// TIA Portal V17 export
// export: Created 2024-08-26T21:07:15.2242134Z, ExportSetting WithDefaults, DisplayName Totally Integrated Automation Portal, DisplayVersion V17 Update 7, DisplayName TIA Portal Openness, DisplayVersion V17 Update 7, DisplayName TIA Portal Version Control Interface, DisplayVersion V17, DisplayName SINAMICS Startdrive Advanced, DisplayVersion V17 SP2, DisplayName SINAMICS Startdrive G110M, G120, G120C, G120D, G120P, G115D, DisplayVersion V17 SP2, DisplayName SINAMICS Startdrive G130, G150, S120, S150, SINAMICS MV, S210, DisplayVersion V17 SP2, DisplayName STEP 7 Professional, DisplayVersion V17 Update 7, DisplayName STEP 7 Safety, DisplayVersion V17 Update 6, DisplayName WinCC Advanced / Unified PC, DisplayVersion V17 Update 7
ORGANIZATION_BLOCK "stationOutputs"   // OB124, LAD, ProgramCycle
TITLE = "Main Program Sweep (Cycle)"
{ S7_Optimized_Access := 'TRUE' }
VERSION : 0.1
// stored: AutoNumber true, IsIECCheckEnabled false, SetENOAutomatically false
   VAR_INPUT
      Initial_Call : Bool;   // Initial call of this OB
      Remanence : Bool;   // =True, if remanent data are available
   END_VAR
BEGIN

REGION Network 1: PRESENT PARTS
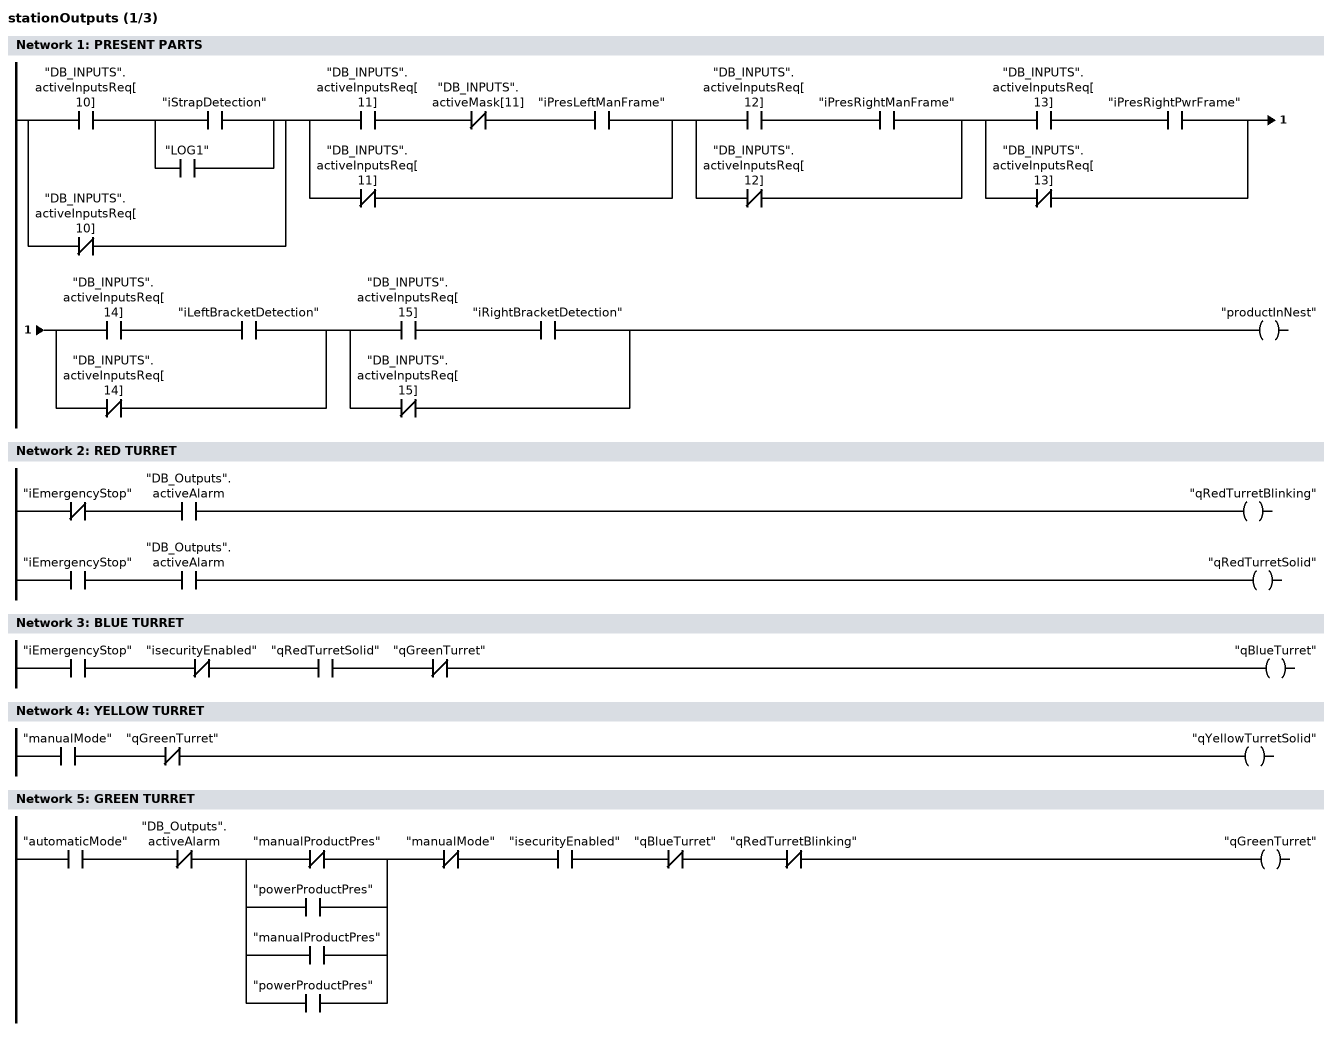
   RUNG wire#powerrail
      Contact( "DB_INPUTS".activeInputsReq[10] )
      wire#w1
      Contact( "iStrapDetection" )
      wire#w2
      Contact( "DB_INPUTS".activeInputsReq[11] )
      I_Contact( "DB_INPUTS".activeMask[11] )
      Contact( "iPresLeftManFrame" )
      wire#w3
      Contact( "DB_INPUTS".activeInputsReq[12] )
      Contact( "iPresRightManFrame" )
      wire#w4
      Contact( "DB_INPUTS".activeInputsReq[13] )
      Contact( "iPresRightPwrFrame" )
      wire#w5
      Contact( "DB_INPUTS".activeInputsReq[14] )
      Contact( "iLeftBracketDetection" )
      wire#w6
      Contact( "DB_INPUTS".activeInputsReq[15] )
      Contact( "iRightBracketDetection" )
      wire#w7
      Coil( "productInNest" )
   END_RUNG
   RUNG wire#w1
      Contact( "LOG1" )
   END_RUNG wire#w2
   RUNG wire#powerrail
      I_Contact( "DB_INPUTS".activeInputsReq[10] )
   END_RUNG wire#w2
   RUNG wire#w2
      I_Contact( "DB_INPUTS".activeInputsReq[11] )
   END_RUNG wire#w3
   RUNG wire#w3
      I_Contact( "DB_INPUTS".activeInputsReq[12] )
   END_RUNG wire#w4
   RUNG wire#w4
      I_Contact( "DB_INPUTS".activeInputsReq[13] )
   END_RUNG wire#w5
   RUNG wire#w5
      I_Contact( "DB_INPUTS".activeInputsReq[14] )
   END_RUNG wire#w6
   RUNG wire#w6
      I_Contact( "DB_INPUTS".activeInputsReq[15] )
   END_RUNG wire#w7
   // the same network as SCL:
   "productInNest" := (("DB_INPUTS".activeInputsReq[10] AND ("iStrapDetection" OR "LOG1")) OR NOT "DB_INPUTS".activeInputsReq[10]) AND (("DB_INPUTS".activeInputsReq[11] AND NOT "DB_INPUTS".activeMask[11] AND "iPresLeftManFrame") OR NOT "DB_INPUTS".activeInputsReq[11]) AND (("DB_INPUTS".activeInputsReq[12] AND "iPresRightManFrame") OR NOT "DB_INPUTS".activeInputsReq[12]) AND (("DB_INPUTS".activeInputsReq[13] AND "iPresRightPwrFrame") OR NOT "DB_INPUTS".activeInputsReq[13]) AND (("DB_INPUTS".activeInputsReq[14] AND "iLeftBracketDetection") OR NOT "DB_INPUTS".activeInputsReq[14]) AND (("DB_INPUTS".activeInputsReq[15] AND "iRightBracketDetection") OR NOT "DB_INPUTS".activeInputsReq[15]);
END_REGION

REGION Network 2: RED TURRET
   RUNG wire#powerrail
      I_Contact( "iEmergencyStop" )
      Contact( "DB_Outputs".activeAlarm )
      Coil( "qRedTurretBlinking" )
   END_RUNG
   RUNG wire#powerrail
      Contact( "iEmergencyStop" )
      Contact( "DB_Outputs".activeAlarm )
      Coil( "qRedTurretSolid" )
   END_RUNG
   // the same network as SCL:
   "qRedTurretBlinking" := NOT "iEmergencyStop" AND "DB_Outputs".activeAlarm;
   "qRedTurretSolid" := "iEmergencyStop" AND "DB_Outputs".activeAlarm;
END_REGION

REGION Network 3: BLUE TURRET
   RUNG wire#powerrail
      Contact( "iEmergencyStop" )
      I_Contact( "isecurityEnabled" )
      Contact( "qRedTurretSolid" )
      I_Contact( "qGreenTurret" )
      Coil( "qBlueTurret" )
   END_RUNG
   // the same network as SCL:
   "qBlueTurret" := "iEmergencyStop" AND NOT "isecurityEnabled" AND "qRedTurretSolid" AND NOT "qGreenTurret";
END_REGION

REGION Network 4: YELLOW TURRET
   RUNG wire#powerrail
      Contact( "manualMode" )
      I_Contact( "qGreenTurret" )
      Coil( "qYellowTurretSolid" )
   END_RUNG
   // the same network as SCL:
   "qYellowTurretSolid" := "manualMode" AND NOT "qGreenTurret";
END_REGION

REGION Network 5: GREEN TURRET
   RUNG wire#powerrail
      Contact( "automaticMode" )
      I_Contact( "DB_Outputs".activeAlarm )
      wire#w1
      I_Contact( "manualProductPres" )
      wire#w2
      I_Contact( "manualMode" )
      Contact( "isecurityEnabled" )
      I_Contact( "qBlueTurret" )
      I_Contact( "qRedTurretBlinking" )
      Coil( "qGreenTurret" )
   END_RUNG
   RUNG wire#w1
      Contact( "powerProductPres" )
   END_RUNG wire#w2
   RUNG wire#w1
      Contact( "manualProductPres" )
   END_RUNG wire#w2
   RUNG wire#w1
      Contact( "powerProductPres" )
   END_RUNG wire#w2
   // the same network as SCL:
   "qGreenTurret" := "automaticMode" AND NOT "DB_Outputs".activeAlarm AND (NOT "manualProductPres" OR "powerProductPres" OR "manualProductPres" OR "powerProductPres") AND NOT "manualMode" AND "isecurityEnabled" AND NOT "qBlueTurret" AND NOT "qRedTurretBlinking";
END_REGION

REGION Network 6: SmartLight
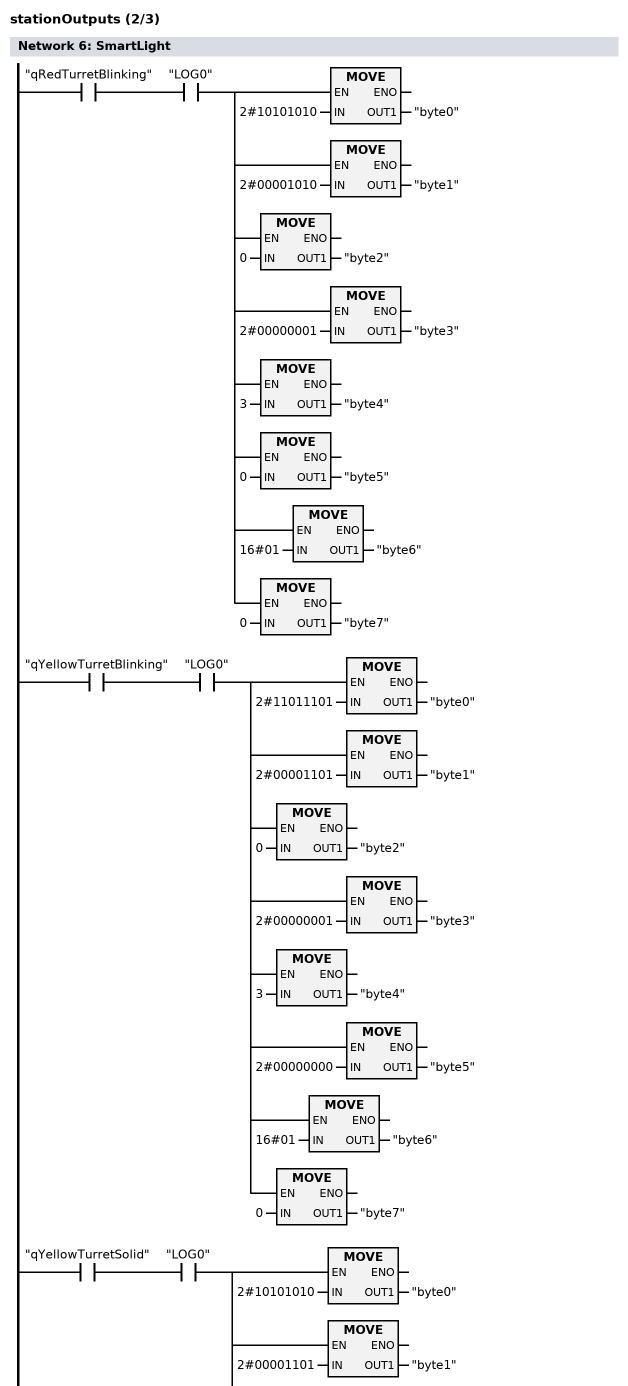
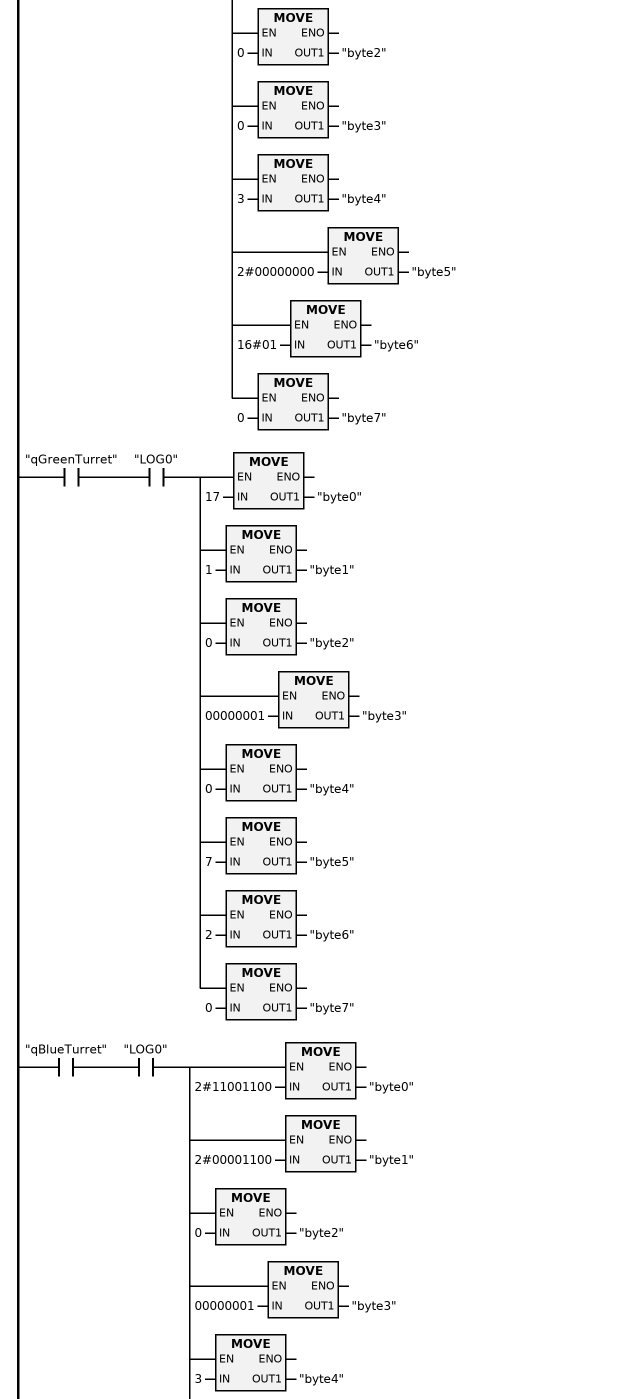
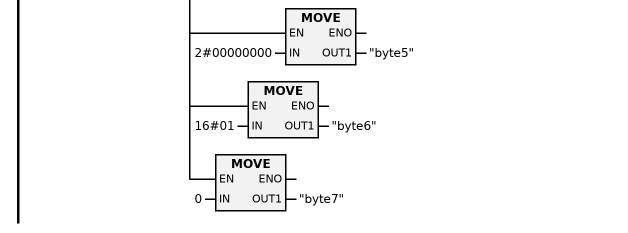
   RUNG wire#powerrail
      Contact( "qRedTurretBlinking" )
      Contact( "LOG0" )
      wire#w1
      Move(in := 2#10101010, out1 => "byte0")
   END_RUNG
   RUNG wire#w1
      Move(in := 2#00001010, out1 => "byte1")
   END_RUNG
   RUNG wire#w1
      Move(in := 0, out1 => "byte2")
   END_RUNG
   RUNG wire#w1
      Move(in := 2#00000001, out1 => "byte3")
   END_RUNG
   RUNG wire#w1
      Move(in := 3, out1 => "byte4")
   END_RUNG
   RUNG wire#w1
      Move(in := 0, out1 => "byte5")
   END_RUNG
   RUNG wire#w1
      Move(in := 16#01, out1 => "byte6")
   END_RUNG
   RUNG wire#w1
      Move(in := 0, out1 => "byte7")
   END_RUNG
   RUNG wire#powerrail
      Contact( "qYellowTurretBlinking" )
      Contact( "LOG0" )
      wire#w2
      Move(in := 2#11011101, out1 => "byte0")
   END_RUNG
   RUNG wire#w2
      Move(in := 2#00001101, out1 => "byte1")
   END_RUNG
   RUNG wire#w2
      Move(in := 0, out1 => "byte2")
   END_RUNG
   RUNG wire#w2
      Move(in := 2#00000001, out1 => "byte3")
   END_RUNG
   RUNG wire#w2
      Move(in := 3, out1 => "byte4")
   END_RUNG
   RUNG wire#w2
      Move(in := 2#00000000, out1 => "byte5")
   END_RUNG
   RUNG wire#w2
      Move(in := 16#01, out1 => "byte6")
   END_RUNG
   RUNG wire#w2
      Move(in := 0, out1 => "byte7")
   END_RUNG
   RUNG wire#powerrail
      Contact( "qYellowTurretSolid" )
      Contact( "LOG0" )
      wire#w3
      Move(in := 2#10101010, out1 => "byte0")
   END_RUNG
   RUNG wire#w3
      Move(in := 2#00001101, out1 => "byte1")
   END_RUNG
   RUNG wire#w3
      Move(in := 0, out1 => "byte2")
   END_RUNG
   RUNG wire#w3
      Move(in := 0, out1 => "byte3")
   END_RUNG
   RUNG wire#w3
      Move(in := 3, out1 => "byte4")
   END_RUNG
   RUNG wire#w3
      Move(in := 2#00000000, out1 => "byte5")
   END_RUNG
   RUNG wire#w3
      Move(in := 16#01, out1 => "byte6")
   END_RUNG
   RUNG wire#w3
      Move(in := 0, out1 => "byte7")
   END_RUNG
   RUNG wire#powerrail
      Contact( "qGreenTurret" )
      Contact( "LOG0" )
      wire#w4
      Move(in := 17, out1 => "byte0")
   END_RUNG
   RUNG wire#w4
      Move(in := 1, out1 => "byte1")
   END_RUNG
   RUNG wire#w4
      Move(in := 0, out1 => "byte2")
   END_RUNG
   RUNG wire#w4
      Move(in := 00000001, out1 => "byte3")
   END_RUNG
   RUNG wire#w4
      Move(in := 0, out1 => "byte4")
   END_RUNG
   RUNG wire#w4
      Move(in := 7, out1 => "byte5")
   END_RUNG
   RUNG wire#w4
      Move(in := 2, out1 => "byte6")
   END_RUNG
   RUNG wire#w4
      Move(in := 0, out1 => "byte7")
   END_RUNG
   RUNG wire#powerrail
      Contact( "qBlueTurret" )
      Contact( "LOG0" )
      wire#w5
      Move(in := 2#11001100, out1 => "byte0")
   END_RUNG
   RUNG wire#w5
      Move(in := 2#00001100, out1 => "byte1")
   END_RUNG
   RUNG wire#w5
      Move(in := 0, out1 => "byte2")
   END_RUNG
   RUNG wire#w5
      Move(in := 00000001, out1 => "byte3")
   END_RUNG
   RUNG wire#w5
      Move(in := 3, out1 => "byte4")
   END_RUNG
   RUNG wire#w5
      Move(in := 2#00000000, out1 => "byte5")
   END_RUNG
   RUNG wire#w5
      Move(in := 16#01, out1 => "byte6")
   END_RUNG
   RUNG wire#w5
      Move(in := 0, out1 => "byte7")
   END_RUNG
   // the same network as SCL:
   IF "qRedTurretBlinking" AND "LOG0" THEN
       "byte0" := 2#10101010;
       "byte1" := 2#00001010;
       "byte2" := 0;
       "byte3" := 2#00000001;
       "byte4" := 3;
       "byte5" := 0;
       "byte6" := 16#01;
       "byte7" := 0;
   END_IF;
   IF "qYellowTurretBlinking" AND "LOG0" THEN
       "byte0" := 2#11011101;
       "byte1" := 2#00001101;
       "byte2" := 0;
       "byte3" := 2#00000001;
       "byte4" := 3;
       "byte5" := 2#00000000;
       "byte6" := 16#01;
       "byte7" := 0;
   END_IF;
   IF "qYellowTurretSolid" AND "LOG0" THEN
       "byte0" := 2#10101010;
       "byte1" := 2#00001101;
       "byte2" := 0;
       "byte3" := 0;
       "byte4" := 3;
       "byte5" := 2#00000000;
       "byte6" := 16#01;
       "byte7" := 0;
   END_IF;
   IF "qGreenTurret" AND "LOG0" THEN
       "byte0" := 17;
       "byte1" := 1;
       "byte2" := 0;
       "byte3" := 00000001;
       "byte4" := 0;
       "byte5" := 7;
       "byte6" := 2;
       "byte7" := 0;
   END_IF;
   IF "qBlueTurret" AND "LOG0" THEN
       "byte0" := 2#11001100;
       "byte1" := 2#00001100;
       "byte2" := 0;
       "byte3" := 00000001;
       "byte4" := 3;
       "byte5" := 2#00000000;
       "byte6" := 16#01;
       "byte7" := 0;
   END_IF;
END_REGION

REGION Network 7: SMART LIGTH CONTROL
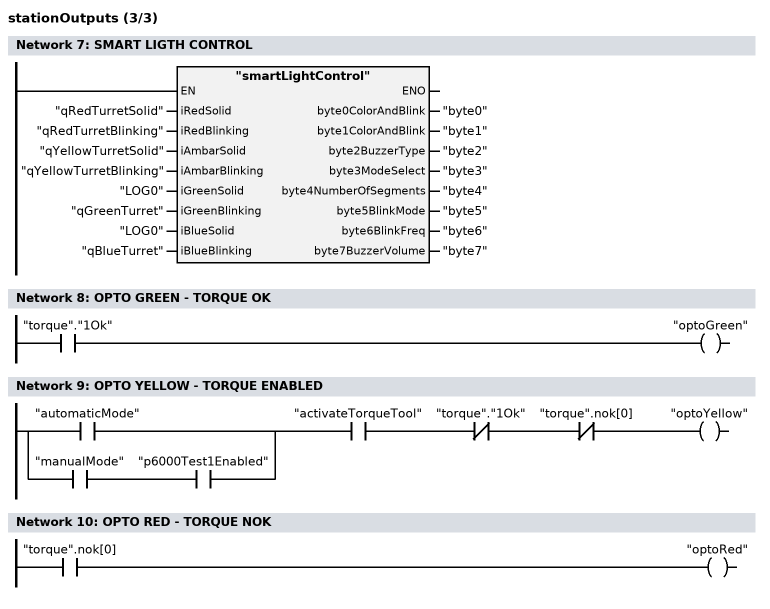
   RUNG wire#powerrail
      "smartLightControl"(iRedSolid := "qRedTurretSolid", iRedBlinking := "qRedTurretBlinking", iAmbarSolid := "qYellowTurretSolid", iAmbarBlinking := "qYellowTurretBlinking", iGreenSolid := "LOG0", iGreenBlinking := "qGreenTurret", iBlueSolid := "LOG0", iBlueBlinking := "qBlueTurret", byte0ColorAndBlink => "byte0", byte1ColorAndBlink => "byte1", byte2BuzzerType => "byte2", byte3ModeSelect => "byte3", byte4NumberOfSegments => "byte4", byte5BlinkMode => "byte5", byte6BlinkFreq => "byte6", byte7BuzzerVolume => "byte7")
   END_RUNG
   // the same network as SCL:
   "smartLightControl"(iRedSolid := "qRedTurretSolid",
                       iRedBlinking := "qRedTurretBlinking",
                       iAmbarSolid := "qYellowTurretSolid",
                       iAmbarBlinking := "qYellowTurretBlinking",
                       iGreenSolid := "LOG0",
                       iGreenBlinking := "qGreenTurret",
                       iBlueSolid := "LOG0",
                       iBlueBlinking := "qBlueTurret",
                       byte0ColorAndBlink => "byte0",
                       byte1ColorAndBlink => "byte1",
                       byte2BuzzerType => "byte2",
                       byte3ModeSelect => "byte3",
                       byte4NumberOfSegments => "byte4",
                       byte5BlinkMode => "byte5",
                       byte6BlinkFreq => "byte6",
                       byte7BuzzerVolume => "byte7");
END_REGION

REGION Network 8: OPTO GREEN - TORQUE OK
   RUNG wire#powerrail
      Contact( "torque"."1Ok" )
      Coil( "optoGreen" )
   END_RUNG
   // the same network as SCL:
   "optoGreen" := "torque"."1Ok";
END_REGION

REGION Network 9: OPTO YELLOW - TORQUE ENABLED
   RUNG wire#powerrail
      Contact( "automaticMode" )
      wire#w1
      Contact( "activateTorqueTool" )
      I_Contact( "torque"."1Ok" )
      I_Contact( "torque".nok[0] )
      Coil( "optoYellow" )
   END_RUNG
   RUNG wire#powerrail
      Contact( "manualMode" )
      Contact( "p6000Test1Enabled" )
   END_RUNG wire#w1
   // the same network as SCL:
   "optoYellow" := ("automaticMode" OR ("manualMode" AND "p6000Test1Enabled")) AND "activateTorqueTool" AND NOT "torque"."1Ok" AND NOT "torque".nok[0];
END_REGION

REGION Network 10: OPTO RED - TORQUE NOK
   RUNG wire#powerrail
      Contact( "torque".nok[0] )
      Coil( "optoRed" )
   END_RUNG
   // the same network as SCL:
   "optoRed" := "torque".nok[0];
END_REGION
END_ORGANIZATION_BLOCK
